FUNCTION_BLOCK FB_2_Skill_SFC EXTENDS FB_1_Skill
VAR_INPUT
	_owner: POINTER TO FB_Base;
	{attribute 'OPC.UA.DA.StructuredType':=1}
	{attribute 'OPC.UA.DA' := '1'}
	Control     : ST_SkillControl;
	{attribute 'OPC.UA.DA.StructuredType':=1}
	{attribute 'OPC.UA.DA' := '1'}
    Status      : ST_SkillStatus;
	Specific	: ST_SkillSpecific;
	SFCInit, SFCPause, SFCReset: BOOL;
END_VAR
VAR_OUTPUT

	SFCError: BOOL;
	SFCCurrentStep: STRING;
END_VAR
VAR

// 	SubSkillHandler : FB_SkillHandler;
END_VAR

ACTION CYCLIC_SFC:
CYCLIC_SKILL();
END_ACTION

METHOD PROTECTED onActivate : eResult
VAR_INPUT
END_VAR

VAR
	eParentResult: eResult;
	myResult: ERESULT;
END_VAR

VAR //YOUR CODE
	succ : BOOL;
END_VAR
eParentResult := SUPER^.onActivate();
//--------------------------------------------------
myResult:=NONE;
// ----- YOUR CODE HERE (incl. Alarms) -------------

myResult:=NONE;

// ----- END YOUR CODE -----------------------------
//--------------------------------------------------
onActivate := CombineResults(eParentResult,myResult);
END_METHOD

METHOD PROTECTED onCleanup : eResult
VAR_INPUT
END_VAR

VAR
	eParentResult: eResult;
	myResult: ERESULT;
END_VAR

VAR //YOUR CODE
	succ : BOOL;
END_VAR
eParentResult := SUPER^.onCleanup();
//--------------------------------------------------
myResult:=NONE;
// ----- YOUR CODE HERE (incl. Alarms) -------------

myResult:=NONE;

// ----- END YOUR CODE -----------------------------
//--------------------------------------------------
onCleanup := CombineResults(eParentResult,myResult);
END_METHOD

METHOD PROTECTED onConfigure : eResult
VAR_INPUT
END_VAR

VAR
	eParentResult: eResult;
	myResult: ERESULT;
END_VAR

VAR //YOUR CODE
	succ : BOOL;
END_VAR
eParentResult := SUPER^.onConfigure();
//--------------------------------------------------
myResult:=NONE;
// ----- YOUR CODE HERE (incl. Alarms) -------------

myResult:=NONE;

// ----- END YOUR CODE -----------------------------
//--------------------------------------------------
onConfigure := CombineResults(eParentResult,myResult);
END_METHOD

METHOD PROTECTED onDeactivate : eResult
VAR_INPUT
END_VAR

VAR
	eParentResult: eResult;
	myResult: ERESULT;
END_VAR

VAR //YOUR CODE
	succ : BOOL;
END_VAR
eParentResult := SUPER^.onDeactivate();
//--------------------------------------------------
myResult:=NONE;
// ----- YOUR CODE HERE (incl. Alarms) -------------

myResult:=NONE;

// ----- END YOUR CODE -----------------------------
//--------------------------------------------------
onDeactivate := CombineResults(eParentResult,myResult);
END_METHOD

METHOD PROTECTED onError : eResult
VAR_INPUT
END_VAR

VAR
	eParentResult: eResult;
	myResult: ERESULT;
END_VAR

VAR //YOUR CODE
	succ : BOOL;
END_VAR
eParentResult := SUPER^.onError();
//--------------------------------------------------
myResult:=NONE;
// ----- YOUR CODE HERE (incl. Alarms) -------------

myResult:=NONE;

// ----- END YOUR CODE -----------------------------
//--------------------------------------------------
onError := CombineResults(eParentResult,myResult);
END_METHOD

METHOD PROTECTED onShutdown : eResult
VAR_INPUT
END_VAR

VAR
	eParentResult: eResult;
	myResult: ERESULT;
END_VAR

VAR //YOUR CODE
	succ : BOOL;
END_VAR
eParentResult := SUPER^.onShutdown();
//--------------------------------------------------
myResult:=NONE;
// ----- YOUR CODE HERE (incl. Alarms) -------------

myResult:=NONE;

// ----- END YOUR CODE -----------------------------
//--------------------------------------------------
onShutdown := CombineResults(eParentResult,myResult);
END_METHOD

END_FUNCTION_BLOCK

(* stored: Version 1.1.0.1, ProductVersion 3.1.4026.18
   POU FB_2_Skill_SFC: Id {bd0554e8-683d-4220-802c-15143a2f2b18}, SpecialFunc None
   Folder StateControl: Id {ed6fe83f-13fc-469d-95a1-90ea828ac04b}
   Action CYCLIC_SFC: Id {fbf93638-4d69-4764-a2ad-53a8ba12e959}
   Method onActivate: Id {e62a8707-006b-4214-80df-3d7118df6453}
   Method onCleanup: Id {1ee1e40f-fc7b-4614-b00d-86d9c771a442}
   Method onConfigure: Id {dc5c12e0-021d-49a1-8746-87ad379a229c}
   Method onDeactivate: Id {2776c250-0af2-41dd-ba5a-bd29717e9f7c}
   Method onError: Id {a254357c-5987-481d-8b51-d3f19aebbf20}
   Method onShutdown: Id {ff585b5e-d6bc-425e-9ccc-ddea2557f2bd} *)
